ABB RobotStudio station: p2_celula_pick&place_R2022.rspag

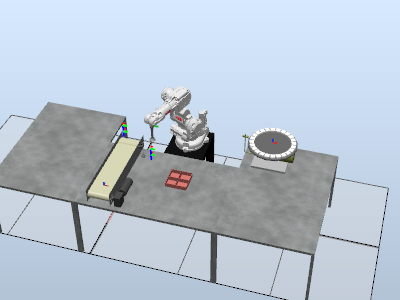
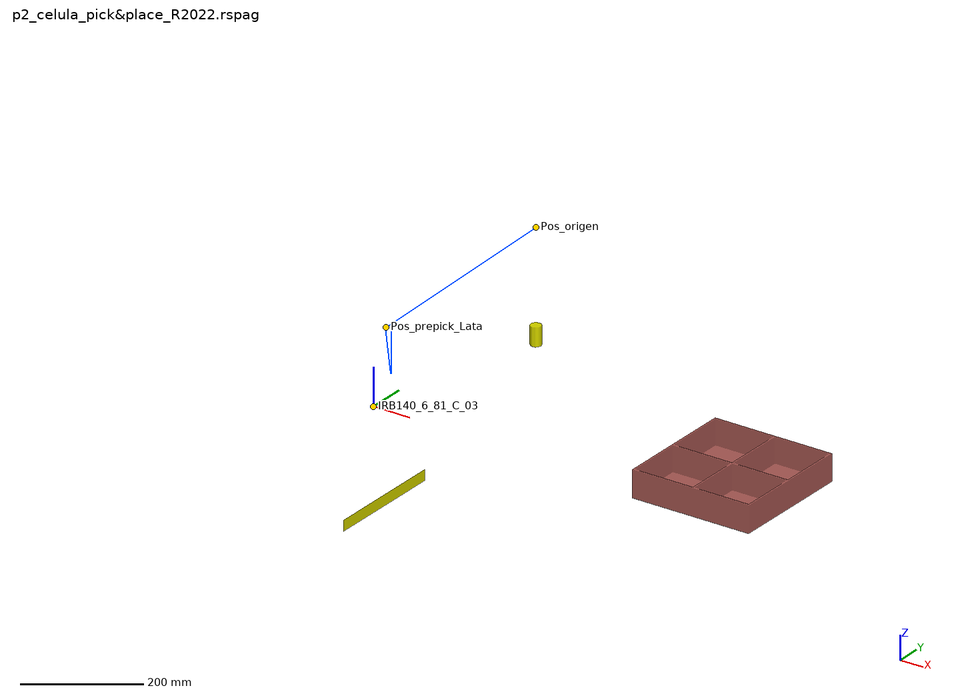
[picture v1: parts stored in the station drawn from their meshes, with robot base, taught points and paths (robot models come from the ABB library and are not in the file)]
--- station ---
Station p2_celula_cinta_mesagir_RS2019_2122_v2 (saved by RobotStudio 22.2.10013.1)
Controller Controlador1, task T_ROB1: task frame (RAPID world) sits at (-250, 750, 760) mm in the station
Controller Controlador1
  mechanical unit ROB_1: IRB140_6_81_C_03, 6 joints, base frame (0, 0, 0) mm
Layout (positions relative to the parent item):
  - Mesa de trabajo [part, from Project\Mesa de trabajo.rslib] at (1000, -110, 0) mm, rotated rx 0 ry 0 rz 90 deg
  - Soporte [part, from Project\SoporteDISA.rslib] at (-500, 970, 0) mm
  - Mesa giratoria [mechanism, from Project\CAD Mesa giratoria.rslib] at (-400, 1510, 760) mm; joint values [1.5268] (rad or m)
  - Mesa de trabajo_2 [part, from Project\Mesa de trabajo_2.rslib] at (1000, 2390, 0) mm, rotated rx 0 ry 0 rz 180 deg
  - cinta_transportadora [smart component, from Project\cinta_transportadoraDISA_RI_vf.rslib]
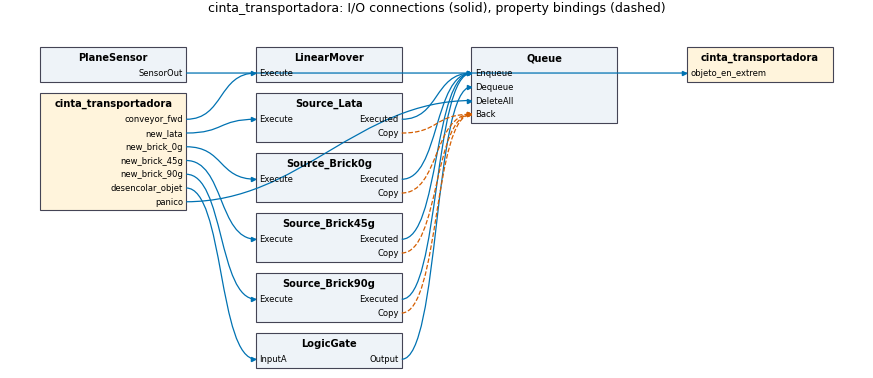
      connections:
        Source_Lata.Executed -> Queue.Enqueue
        PlaneSensor.SensorOut -> cinta_transportadora.objeto_en_extremo
        LogicGate.Output -> Queue.Dequeue
        cinta_transportadora.conveyor_fwd -> LinearMover.Execute
        cinta_transportadora.new_lata -> Source_Lata.Execute
        cinta_transportadora.new_brick_0g -> Source_Brick0g.Execute
        Source_Brick0g.Executed -> Queue.Enqueue
        cinta_transportadora.new_brick_45g -> Source_Brick45g.Execute
        Source_Brick45g.Executed -> Queue.Enqueue
        cinta_transportadora.new_brick_90g -> Source_Brick90g.Execute
        Source_Brick90g.Executed -> Queue.Enqueue
        cinta_transportadora.desencolar_objeto -> LogicGate.InputA
        cinta_transportadora.panico -> Queue.DeleteAll
        Source_Lata.Copy => Queue.Back
        Source_Brick0g.Copy => Queue.Back
        Source_Brick45g.Copy => Queue.Back
        Source_Brick90g.Copy => Queue.Back
    - Cinta transportadora [mechanism, from Project\CAD Cinta transportadora_2.rslib] at (940, 100, 865) mm, rotated rx 0 ry 0 rz 90 deg; joint values [0.66] (rad or m)
    - PlaneSensor [smart component, from Components\PlaneSensor.rslib]
        properties: Origin=[0.17366 0.29 0.93]; Axis1=[0 -0.23 0]; Axis2=[0 0 0.02]; SensedPart=(none)
      - _sensorPart_ [part], size 0 x 230 x 20 mm
    - Source_Lata [smart component, from Components\Source.rslib]
        properties: Source=lata_v3; Copy=(none); Parent=(none); Position=[0.9 0.175 0.9]; Orientation=[0 0 0]; Transient=false; PhysicsBehavior=0
    - Queue [smart component, from Components\Queue.rslib]
        properties: Back=(none); Front=(none); Queue={dff8c8d8-8fc0-4cec-b9db-be29e3a28473};{3f46c5cd-6d5b-48fe-86d8-48bb79a4d1fd};{fed15a07-9f68-4789-ad83-d232714e4fef};{72d5c8a9-7ca8-44e4-9c22-05c1b903e3c3};{2c04b273-edbc-4b62-af70-7d1944a2b1a7};{dd89b5b9-4857-4fa3-833c-eec227f403e2};{f4eddf35-6998-4428-b7c9-fa89e61066a5};{59d38785-21a3-4095-b70c-dd76d22c82fa};{f58c88b0-8b1a-4677-834d-2538b4835fbc};{bf0dbb8d-c78c-4188-b692-762c5a23a001};{d95e0b15-e936-410f-9e61-fe724db3c540};{2bd839ac-2019-415b-83b6-f6b4b81f6058};{944dfd5c-fb13-4575-94b9-afd36fb7f782};{83949a1e-8185-4c93-aa89-25b66602ceee};{4f3442c7-6ec6-4cb3-811a-33626f372c7a};{e17365bb-1bef-470b-b7e8-ca19aadd4809};{cf2dd58a-cd53-48dc-b704-49735820749d};{8950a759-9402-4139-8874-5414b657c79d};{ff666c08-3b55-4b31-af91-fb9ccf20597e};{00479655-b269-4748-adfd-ac0c9ff6814e};{97aee651-0048-42db-8271-c3c0405e84b6};{fb9d78cf-dec4-43c5-9643-90b43aa2c589};{1c737023-80b2-404b-b5f7-6a789b37bf94};{1ad73b80-f19d-4287-9cc4-3f5d513c44b3};{4a9cfcbd-6104-4fda-bb66-45b7a58cadba};{f5030ce7-8d9f-41fd-a0e0-943b87f40044};{6d643d8b-3f64-40eb-a316-e6579e800488};{a521ad28-28eb-4a02-9bff-ecd8140946c6};{54e7b961-4a7e-4eb9-9ad8-12fd860b0d09};{a76ff4cc-00e3-4c57-a249-5d676800b108};{a962051d-4321-485d-a7b6-d46c092dbce2};{12afaf56-49c6-4ccb-a620-f61642ea87b3};{899343f8-8cec-4edb-8463-23c64231605d};{4ef6d4c1-cd94-4d60-a742-53b60612dce5};{81835927-5480-4704-8e95-458aff66f5f4};{f557f8d3-d4c2-4ed9-81ee-a7371f7a9064};{a3283dab-8ae5-4a2f-a5f1-e3aa67324f00};{c73702e9-d765-4ca0-822f-348813278423};{414af213-d7ca-4e68-bc40-e9049d23ee9f};{a443fb2b-66d5-488a-b1cc-adbb6ebe2bc4};{96543467-7996-4e03-8609-ae8e4ea8f5a5};{8d69ce69-ef13-48be-9f25-6767b80184bb};{3789e405-e3ee-43e3-9d44-f2b54c75a36d};{dcf48f4d-3edb-45db-ad86-a5594296e2e2};{558120a7-5c88-4567-bb6c-c613c49afc30};{e83fdc9f-8db8-4194-8e9e-23232cbce353};{e901d7c8-de42-4474-a4d8-69454c384dc7};{2ec176ed-b9bc-4276-a128-5d5885d6c924};{8a74c292-b841-49af-a904-a0eec89b4ec6};{28ce9f31-519e-4f33-90fc-d50f408da8a6};{7a6d8f97-5379-4c1c-bdf6-f3c9a7aad7fa};{93e37ce4-f8bb-47c1-a0d2-06e10bf97d3f};{e8c5fbea-3965-4645-a5b7-c30112c44e96};{e7a5134e-a405-458e-8997-754f0378309b};{c78df5ee-6dfc-4a92-ba12-8dbc026209cf};{b1b4c00c-25a8-4bd7-80e1-6afde583105d};{dd0c4c06-6ce6-4be1-9c99-64db0c6bf6ff};{cefc24b7-ae8e-4a04-b8e7-f81f9433e3ae};{d6ce0fe5-35b2-42bb-b8d6-adbba0a8763d};{632131fa-8e51-4513-abd4-76a5ea6fcb33};{74bd1469-f266-4be2-92ac-ab91072705d8};{f6b76230-9575-465d-b1fa-b377b73fd13a};{9029fc77-8703-416f-ba68-5dca8c19555c};{b0ece3da-778c-4de5-ae49-5dd73d9e5191};{a4b8dd9f-1cea-46ee-b3db-e7479fcd6562};{ef382f55-caa7-4132-9e3f-cf775111e149};{7208aa9c-0a4c-4c08-824b-10d06152fb4f};{56b747bb-a3fb-4c38-b62b-aa802f47d477};{eb7448c0-cf7b-415d-9783-7e65fa723709};{f3dda0a0-cbf2-45ab-a7de-e8869eedcb74}; NumberOfObjects=0
    - LogicGate [smart component, from Components\LogicGate.rslib]
        properties: Operator=NOT; Delay=0
    - LinearMover [smart component, from Components\LinearMover.rslib]
        properties: Object=Queue; Direction=[1 0 0]; Speed=-0.1; Reference=Global; ReferenceObject=(none)
    - Source_Brick0g [smart component, from Components\Source.rslib]
        properties: Source=Brick0g; Copy=(none); Parent=(none); Position=[0.7 0.13 0.9]; Orientation=[0 0 0]; Transient=false; PhysicsBehavior=0
    - Source_Brick45g [smart component, from Components\Source.rslib]
        properties: Source=Brick0g; Copy=(none); Parent=(none); Position=[0.77 0.08 0.9]; Orientation=[0 0 0.785398163397448]; Transient=false; PhysicsBehavior=0
    - Source_Brick90g [smart component, from Components\Source.rslib]
        properties: Source=Brick0g; Copy=(none); Parent=(none); Position=[0.93 0.065 0.9]; Orientation=[0 0 1.5707963267949]; Transient=false; PhysicsBehavior=0
  - Pieza_11 [part], size 231 x 233 x 51.1 mm
  - Mesa de trabajo_3 [part, from Project\Mesa de trabajo_3.rslib] at (1000, -110, 0) mm, rotated rx 0 ry 0 rz 180 deg
  - ventosa_giu [smart component, from Project\ventosa_DISA_RI.rslib] at (245, 500, 1320) mm, rotated rx 180 ry 0 rz -180 deg
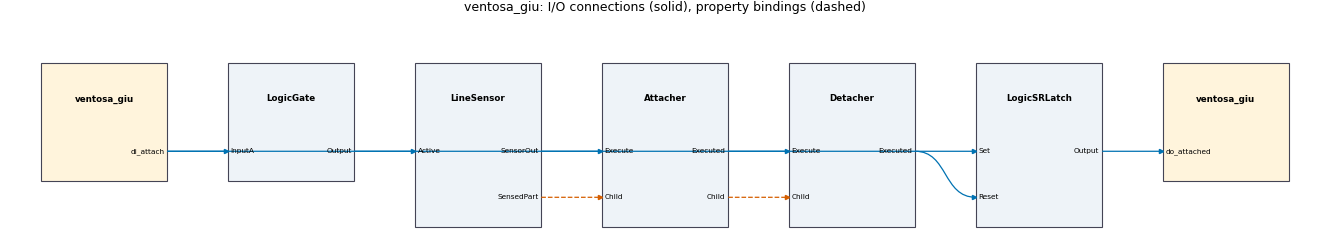
      connections:
        ventosa_giu.di_attach -> LogicGate.InputA
        LineSensor.SensorOut -> Attacher.Execute
        LogicGate.Output -> LineSensor.Active
        ventosa_giu.di_attach -> Detacher.Execute
        Attacher.Executed -> LogicSRLatch.Set
        Detacher.Executed -> LogicSRLatch.Reset
        LogicSRLatch.Output -> ventosa_giu.do_attached
        LineSensor.SensedPart => Attacher.Child
        Attacher.Child => Detacher.Child
    - ventosa_disa_giu [part, from Project\ventosa_DISA_RI.rslib]
    - LogicGate [smart component, from Components\LogicGate.rslib]
        properties: Operator=NOT; Delay=0
    - LineSensor [smart component, from Components\LineSensor.rslib]
        properties: Start=[0 0 0.175]; End=[0 0 0.21]; Radius=0.01; SensedPart=(none); SensedPoint=[0.337000091552734 0.776 0.848742248535156]
      - _sensorPart_ [part], size 20 x 20 x 35 mm
    - Attacher [smart component, from Components\Attacher.rslib]
        properties: Parent=ventosa_giu; Flange=0; Child=(none); Mount=false; Offset=[0 0 0]; Orientation=[0 0 0]
    - Detacher [smart component, from Components\Detacher.rslib]
        properties: Child=(none); KeepPosition=true
    - LogicSRLatch [smart component, from Components\LogicSRLatch.rslib]
  - IRB140_6_81_C_03 [mechanism, from Robots\IRB140_6_81_C_G_03.rslib] at (-250, 750, 760) mm; joint values [-0.4677, 0.3133, -0.1294, 0, 1.3869, -0.4677] (rad or m)
  - Brick0g [part], size 215 x 90 x 69 mm
  - lata_v3 [part], size 96.5 x 96.5 x 81.4 mm
Attachment: ventosa_giu is attached to IRB140_6_81_C_03 / Link6
EventTableEntry 9242: Group=, Trigger=Abrir 9243, Actions=[EventTableActionNothing 12035, EventTableActionDetach 12036, EventTableActionDetach 12037, EventTableActionDetach 12038, EventTableActionDetach 12039, EventTableActionDetach 12040, EventTableActionDetach 12041], Comment=, ActivationMode=2, Cyclic=true
EventTableTriggerIO 9243: IOValue=[1], IRC5Controller=? -1, Operator=0, SignalSource=? -1
EventTableEntry 9251: Group=, Trigger=Cerrar 9252, Actions=[EventTableActionDetach 12042, EventTableActionDetach 12043, EventTableActionDetach 12044, EventTableActionDetach 12045, EventTableActionDetach 12046, EventTableActionDetach 12047, EventTableActionNothing 12048], Comment=, ActivationMode=2, Cyclic=true
EventTableTriggerIO 9252: IOValue=[1], IRC5Controller=? -1, Operator=0, SignalSource=? -1
EventTableEntry 9264: Group=, Trigger=NOP 9265, Actions=[Abrir 9267], Comment=, ActivationMode=2, Cyclic=false
EventTableTriggerLogic 9265: Operand1=DoGARRAOPEN 9266, Operand2=? -1, Operator=4, Delay=1000
EventTableTriggerIO 9266: IOValue=[-1], IRC5Controller=? -1, Operator=0, SignalSource=? -1
EventTableActionIO 9267: IOValue=[-1], IRC5Controller=? -1, SignalTarget=? -1
EventTableEntry 9268: Group=, Trigger=NOT 9269, Actions=[Cerrar 9271], Comment=, ActivationMode=2, Cyclic=false
EventTableTriggerLogic 9269: layoutX=105, layoutY=91, Operand1=DoGARRAOPEN 9270, Operand2=? -1, Operator=2, Delay=1000
EventTableTriggerIO 9270: IOValue=[-1], IRC5Controller=? -1, Operator=0, SignalSource=? -1
EventTableActionIO 9271: IOValue=[-1], IRC5Controller=? -1, SignalTarget=? -1
EventTableEntry 9272: Group=, Trigger=DoGARRAOPEN 9273, Actions=[EventTableActionMechanicalPose 9274], Comment=, ActivationMode=2, Cyclic=false
EventTableTriggerIO 9273: IOValue=[1], IRC5Controller=? -1, Operator=0, SignalSource=? -1
EventTableActionMechanicalPose 9274: VirtualSignal=, Mechanism=? -1, ToPoseName=Abierta, VirtualSignalValue=[1]
EventTableEntry 9275: Group=, Trigger=DoGARRAOPEN 9276, Actions=[EventTableActionMechanicalPose 9277], Comment=, ActivationMode=2, Cyclic=false
EventTableTriggerIO 9276: IOValue=[0], IRC5Controller=? -1, Operator=0, SignalSource=? -1
EventTableActionMechanicalPose 9277: VirtualSignal=, Mechanism=? -1, ToPoseName=Cerrada, VirtualSignalValue=[1]
EventTableEntry 9288: Group=, Trigger=DO10_4 9289, Actions=[EventTableActionMechanicalPose 10691, EventTableActionMechanicalPose 10690, EventTableActionMechanicalPose 10689, EventTableActionMechanicalPose 11250, EventTableActionMechanicalPose 11251, EventTableActionMechanicalPose 11252], Comment=, ActivationMode=2, Cyclic=true
EventTableTriggerIO 9289: IOValue=[1], IRC5Controller=? -1, Operator=0, SignalSource=? -1
EventTableEntry 9711: Group=, Trigger=Abrir 9712, Actions=[EventTableActionNothing 12049, EventTableActionAttach 12050, EventTableActionAttach 12051, EventTableActionAttach 12052, EventTableActionNothing 12053, EventTableActionNothing 12054, EventTableActionNothing 12055], Comment=, ActivationMode=2, Cyclic=true
EventTableTriggerIO 9712: IOValue=[1], IRC5Controller=? -1, Operator=0, SignalSource=? -1
EventTableEntry 9938: Group=, Trigger=Cerrar 9939, Actions=[EventTableActionAttach 12056, EventTableActionAttach 12057, EventTableActionAttach 12058, EventTableActionAttach 12059, EventTableActionAttach 12060, EventTableActionAttach 12061, EventTableActionNothing 12062], Comment=, ActivationMode=2, Cyclic=true
EventTableTriggerIO 9939: IOValue=[1], IRC5Controller=? -1, Operator=0, SignalSource=? -1
EventTableActionMechanicalPose 10689: VirtualSignal=, Mechanism=Mesa giratoria 10339, ToPoseName=360º, VirtualSignalValue=[1]
EventTableActionMechanicalPose 10690: VirtualSignal=, Mechanism=Mesa giratoria 10339, ToPoseName=180º, VirtualSignalValue=[1]
EventTableActionMechanicalPose 10691: VirtualSignal=, Mechanism=Mesa giratoria 10339, ToPoseName=90º, VirtualSignalValue=[1]
EventTableEntry 11031: Group=, Trigger=DO10_5 11032, Actions=[EventTableActionAttach 11212, EventTableActionAttach 11213, EventTableActionAttach 11214], Comment=, ActivationMode=2, Cyclic=true
EventTableTriggerIO 11032: IOValue=[1], IRC5Controller=? -1, Operator=0, SignalSource=? -1
EventTableEntry 11051: Group=, Trigger=Abrir 11052, Actions=[EventTableActionNothing 12063, EventTableActionMechanicalPose 12064, EventTableActionMechanicalPose 12065, EventTableActionNothing 12066, EventTableActionNothing 12067, EventTableActionNothing 12068, EventTableActionNothing 12069], Comment=, ActivationMode=2, Cyclic=true
EventTableTriggerIO 11052: IOValue=[1], IRC5Controller=? -1, Operator=0, SignalSource=? -1
EventTableEntry 11203: Group=, Trigger=DO10_5 11204, Actions=[EventTableActionMechanicalPose 11205, EventTableActionMechanicalPose 11206, EventTableActionMechanicalPose 11207], Comment=, ActivationMode=2, Cyclic=true
EventTableTriggerIO 11204: IOValue=[1], IRC5Controller=? -1, Operator=0, SignalSource=? -1
EventTableActionMechanicalPose 11205: VirtualSignal=, Mechanism=Cinta transportadora 10989, ToPoseName=HomePosition, VirtualSignalValue=[1]
EventTableActionMechanicalPose 11206: VirtualSignal=, Mechanism=Cinta transportadora 10989, ToPoseName=HomePosition, VirtualSignalValue=[1]
EventTableActionMechanicalPose 11207: VirtualSignal=, Mechanism=Cinta transportadora 10989, ToPoseName=HomePosition, VirtualSignalValue=[1]
EventTableActionAttach 11212: AttachmentParent=Cinta transportadora 10989, AttachmentChild=? -1, MountObject=false, Offset=[X=1, Y=0, Z=0, W=0, X=0, Y=1, Z=0, W=0, X=0, Y=0, Z=1, W=0, X=0, Y=0, Z=0, W=1], FlangeIndext=0, FindNearest=false
EventTableActionAttach 11213: AttachmentParent=Cinta transportadora 10989, AttachmentChild=? -1, MountObject=false, Offset=[X=1, Y=0, Z=0, W=0, X=0, Y=1, Z=0, W=0, X=0, Y=0, Z=1, W=0, X=0, Y=0, Z=0, W=1], FlangeIndext=0, FindNearest=false
EventTableActionAttach 11214: AttachmentParent=Cinta transportadora 10989, AttachmentChild=? -1, MountObject=false, Offset=[X=1, Y=0, Z=0, W=0, X=0, Y=1, Z=0, W=0, X=0, Y=0, Z=1, W=0, X=0, Y=0, Z=0, W=1], FlangeIndext=0, FindNearest=false
EventTableActionMechanicalPose 11250: VirtualSignal=, Mechanism=Mesa giratoria 10339, ToPoseName=450, VirtualSignalValue=[1]
EventTableActionMechanicalPose 11251: VirtualSignal=, Mechanism=Mesa giratoria 10339, ToPoseName=540º, VirtualSignalValue=[1]
EventTableActionMechanicalPose 11252: VirtualSignal=, Mechanism=Mesa giratoria 10339, ToPoseName=SyncPosition, VirtualSignalValue=[1]
EventTableEntry 11270: Group=, Trigger=DO10_6 11271, Actions=[EventTableActionAttach 11272, EventTableActionAttach 11273, EventTableActionAttach 11274], Comment=, ActivationMode=2, Cyclic=true
EventTableTriggerIO 11271: IOValue=[1], IRC5Controller=? -1, Operator=0, SignalSource=? -1
EventTableActionAttach 11272: AttachmentParent=Cinta transportadora 10989, AttachmentChild=? -1, MountObject=false, Offset=[X=1, Y=0, Z=0, W=0, X=0, Y=1, Z=0, W=0, X=0, Y=0, Z=1, W=0, X=0, Y=0, Z=0, W=1], FlangeIndext=0, FindNearest=false
EventTableActionAttach 11273: AttachmentParent=Cinta transportadora 10989, AttachmentChild=? -1, MountObject=false, Offset=[X=1, Y=0, Z=0, W=0, X=0, Y=1, Z=0, W=0, X=0, Y=0, Z=1, W=0, X=0, Y=0, Z=0, W=1], FlangeIndext=0, FindNearest=false
EventTableActionAttach 11274: AttachmentParent=Cinta transportadora 10989, AttachmentChild=? -1, MountObject=false, Offset=[X=1, Y=0, Z=0, W=0, X=0, Y=1, Z=0, W=0, X=0, Y=0, Z=1, W=0, X=0, Y=0, Z=0, W=1], FlangeIndext=0, FindNearest=false
EventTableEntry 11487: Group=, Trigger=Cerrar 11488, Actions=[EventTableActionNothing 12070, EventTableActionNothing 12071, EventTableActionNothing 12072, EventTableActionNothing 12073, EventTableActionMechanicalPose 12074, EventTableActionMechanicalPose 12075, EventTableActionNothing 12076], Comment=, ActivationMode=2, Cyclic=true
EventTableTriggerIO 11488: IOValue=[1], IRC5Controller=? -1, Operator=0, SignalSource=? -1
EventTableEntry 11751: Group=, Trigger=Cerrar 11752, Actions=[EventTableActionNothing 12077, EventTableActionNothing 12078, EventTableActionNothing 12079, EventTableActionNothing 12080, EventTableActionDetach 12081, EventTableActionDetach 12082, EventTableActionDetach 12083], Comment=, ActivationMode=2, Cyclic=true
EventTableTriggerIO 11752: IOValue=[1], IRC5Controller=? -1, Operator=0, SignalSource=? -1
EventTableEntry 11847: Group=, Trigger=DO10_6 11848, Actions=[EventTableActionMechanicalPose 11849, EventTableActionMechanicalPose 11850, EventTableActionMechanicalPose 11851], Comment=, ActivationMode=2, Cyclic=true
EventTableTriggerIO 11848: IOValue=[1], IRC5Controller=? -1, Operator=0, SignalSource=? -1
EventTableActionMechanicalPose 11849: VirtualSignal=, Mechanism=Cinta transportadora 10989, ToPoseName=Final, VirtualSignalValue=[1]
EventTableActionMechanicalPose 11850: VirtualSignal=, Mechanism=Cinta transportadora 10989, ToPoseName=Final, VirtualSignalValue=[1]
EventTableActionMechanicalPose 11851: VirtualSignal=, Mechanism=Cinta transportadora 10989, ToPoseName=Final, VirtualSignalValue=[1]
EventTableActionNothing 12035: 
EventTableActionDetach 12036: AttachmentParent=? -1, AttachmentChild=? -1
EventTableActionDetach 12037: AttachmentParent=? -1, AttachmentChild=? -1
EventTableActionDetach 12038: AttachmentParent=? -1, AttachmentChild=? -1
EventTableActionDetach 12039: AttachmentParent=? -1, AttachmentChild=? -1
EventTableActionDetach 12040: AttachmentParent=? -1, AttachmentChild=? -1
EventTableActionDetach 12041: AttachmentParent=? -1, AttachmentChild=? -1
EventTableActionDetach 12042: AttachmentParent=Cinta transportadora 10989, AttachmentChild=? -1
EventTableActionDetach 12043: AttachmentParent=Cinta transportadora 10989, AttachmentChild=? -1
EventTableActionDetach 12044: AttachmentParent=Cinta transportadora 10989, AttachmentChild=? -1
EventTableActionDetach 12045: AttachmentParent=Mesa giratoria 10339, AttachmentChild=? -1
EventTableActionDetach 12046: AttachmentParent=Mesa giratoria 10339, AttachmentChild=? -1
EventTableActionDetach 12047: AttachmentParent=Mesa giratoria 10339, AttachmentChild=? -1
EventTableActionNothing 12048: 
EventTableActionNothing 12049: 
EventTableActionAttach 12050: AttachmentParent=Mesa giratoria 10339, AttachmentChild=? -1, MountObject=false, Offset=[X=1, Y=0, Z=0, W=0, X=0, Y=1, Z=0, W=0, X=0, Y=0, Z=1, W=0, X=0, Y=0, Z=0, W=1], FlangeIndext=0, FindNearest=false
EventTableActionAttach 12051: AttachmentParent=Mesa giratoria 10339, AttachmentChild=? -1, MountObject=false, Offset=[X=1, Y=0, Z=0, W=0, X=0, Y=1, Z=0, W=0, X=0, Y=0, Z=1, W=0, X=0, Y=0, Z=0, W=1], FlangeIndext=0, FindNearest=false
EventTableActionAttach 12052: AttachmentParent=Mesa giratoria 10339, AttachmentChild=? -1, MountObject=false, Offset=[X=1, Y=0, Z=0, W=0, X=0, Y=1, Z=0, W=0, X=0, Y=0, Z=1, W=0, X=0, Y=0, Z=0, W=1], FlangeIndext=0, FindNearest=false
EventTableActionNothing 12053: 
EventTableActionNothing 12054: 
EventTableActionNothing 12055: 
EventTableActionAttach 12056: AttachmentParent=? -1, AttachmentChild=? -1, MountObject=true, Offset=[X=1, Y=0, Z=0, W=0, X=0, Y=1, Z=0, W=0, X=0, Y=0, Z=1, W=0, X=0, Y=0, Z=0, W=1], FlangeIndext=0, FindNearest=false
EventTableActionAttach 12057: AttachmentParent=? -1, AttachmentChild=? -1, MountObject=true, Offset=[X=1, Y=0, Z=0, W=0, X=0, Y=1, Z=0, W=0, X=0, Y=0, Z=1, W=0, X=0, Y=0, Z=0, W=1], FlangeIndext=0, FindNearest=false
EventTableActionAttach 12058: AttachmentParent=? -1, AttachmentChild=? -1, MountObject=true, Offset=[X=1, Y=0, Z=0, W=0, X=0, Y=1, Z=0, W=0, X=0, Y=0, Z=1, W=0, X=0, Y=0, Z=0, W=1], FlangeIndext=0, FindNearest=false
EventTableActionAttach 12059: AttachmentParent=? -1, AttachmentChild=? -1, MountObject=true, Offset=[X=1, Y=0, Z=0, W=0, X=0, Y=1, Z=0, W=0, X=0, Y=0, Z=1, W=0, X=0, Y=0, Z=0, W=1], FlangeIndext=0, FindNearest=false
EventTableActionAttach 12060: AttachmentParent=? -1, AttachmentChild=? -1, MountObject=true, Offset=[X=1, Y=0, Z=0, W=0, X=0, Y=1, Z=0, W=0, X=0, Y=0, Z=1, W=0, X=0, Y=0, Z=0, W=1], FlangeIndext=0, FindNearest=false
EventTableActionAttach 12061: AttachmentParent=? -1, AttachmentChild=? -1, MountObject=true, Offset=[X=1, Y=0, Z=0, W=0, X=0, Y=1, Z=0, W=0, X=0, Y=0, Z=1, W=0, X=0, Y=0, Z=0, W=1], FlangeIndext=0, FindNearest=false
EventTableActionNothing 12062: 
EventTableActionNothing 12063: 
EventTableActionMechanicalPose 12064: VirtualSignal=, Mechanism=Cinta transportadora 10989, ToPoseName=Final_2, VirtualSignalValue=[1]
EventTableActionMechanicalPose 12065: VirtualSignal=, Mechanism=Cinta transportadora 10989, ToPoseName=Final_2, VirtualSignalValue=[1]
EventTableActionNothing 12066: 
EventTableActionNothing 12067: 
EventTableActionNothing 12068: 
EventTableActionNothing 12069: 
EventTableActionNothing 12070: 
EventTableActionNothing 12071: 
EventTableActionNothing 12072: 
EventTableActionNothing 12073: 
EventTableActionMechanicalPose 12074: VirtualSignal=, Mechanism=Cinta transportadora 10989, ToPoseName=Pose inicial_2, VirtualSignalValue=[1]
EventTableActionMechanicalPose 12075: VirtualSignal=, Mechanism=Cinta transportadora 10989, ToPoseName=Pose inicial_2, VirtualSignalValue=[1]
EventTableActionNothing 12076: 
EventTableActionNothing 12077: 
EventTableActionNothing 12078: 
EventTableActionNothing 12079: 
EventTableActionNothing 12080: 
EventTableActionDetach 12081: AttachmentParent=Cinta transportadora 10989, AttachmentChild=? -1
EventTableActionDetach 12082: AttachmentParent=Cinta transportadora 10989, AttachmentChild=? -1
EventTableActionDetach 12083: AttachmentParent=Cinta transportadora 10989, AttachmentChild=? -1
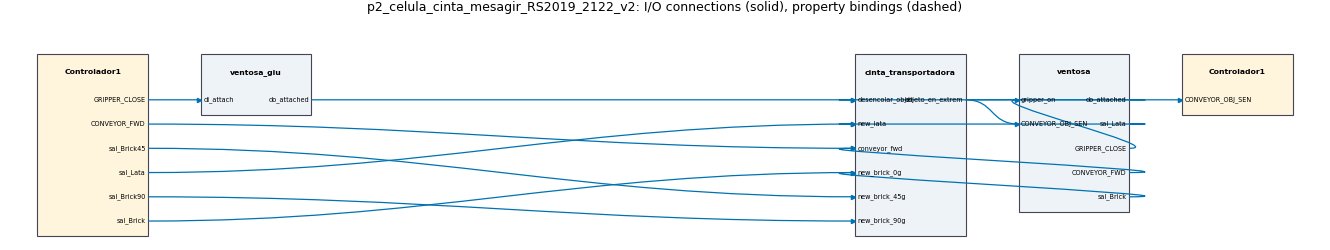
Station logic (signal -> signal, property => property):
  ventosa.do_attached -> cinta_transportadora.desencolar_objeto
  Controlador_P2_2021.sal_Lata -> cinta_transportadora.new_lata
  Controlador_P2_2021.GRIPPER_CLOSE -> ventosa.gripper_on
  cinta_transportadora.objeto_en_extremo -> Controlador_P2_2021.CONVEYOR_OBJ_SEN
  Controlador_P2_2021.CONVEYOR_FWD -> cinta_transportadora.conveyor_fwd
  Controlador_P2_2021.sal_Brick -> cinta_transportadora.new_brick_0g
  Controlador1.GRIPPER_CLOSE -> ventosa_giu.di_attach
  Controlador1.CONVEYOR_FWD -> cinta_transportadora.conveyor_fwd
  Controlador1.sal_Brick45 -> cinta_transportadora.new_brick_45g
  Controlador1.sal_Lata -> cinta_transportadora.new_lata
  Controlador1.sal_Brick90 -> cinta_transportadora.new_brick_90g
  Controlador1.sal_Brick -> cinta_transportadora.new_brick_0g
  cinta_transportadora.objeto_en_extremo -> Controlador1.CONVEYOR_OBJ_SEN
  ventosa_giu.do_attached -> cinta_transportadora.desencolar_objeto

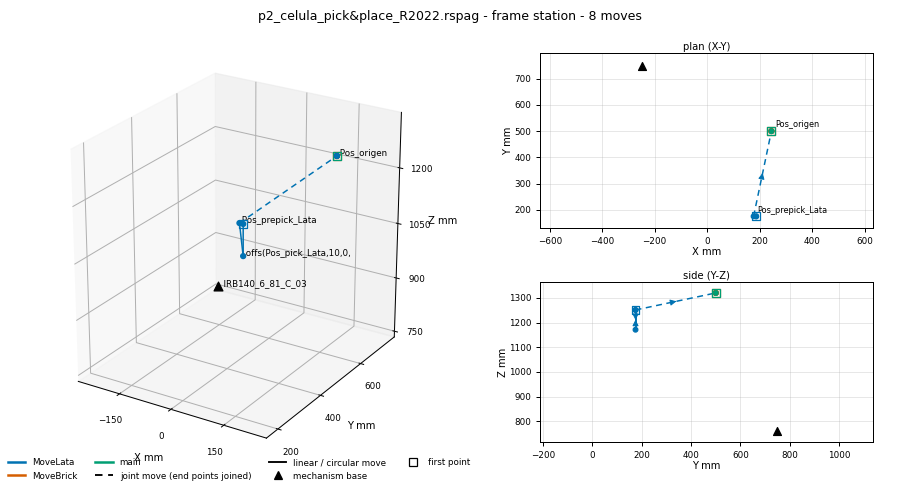
[picture p0: tool path of p2_celula_pick&place_R2022.rspag in frame station, 8 of 18 moves have a stored position in this frame; points joined in program order, loops and branches not executed]
--- Backups/Controlador1/RAPID/TASK1/PROGMOD/MainModule.mod ---
MODULE MainModule

    FUNC orient quatProd(orient o1, orient o2)


        RETURN [
            o1.q1 * o2.q1 - o1.q2 * o2.q2 - o1.q3 * o2.q3 - o1.q4 * o2.q4,
            o1.q1 * o2.q2 + o1.q2 * o2.q1 + o1.q3 * o2.q4 - o1.q4 * o2.q3,
            o1.q1 * o2.q3 + o1.q3 * o2.q1 + o1.q4 * o2.q2 - o1.q2 * o2.q4,
            o1.q1 * o2.q4 + o1.q4 * o2.q1 + o1.q2 * o2.q3 - o1.q3 * o2.q2];
    ENDFUNC


    PROC MoveLata(num latas,num layer)
        VAR robtarget preplace := Pos_preplace_lata;
        VAR robtarget place := Pos_place_lata;


        MoveL offs(Pos_prepick_Lata,10,0,0), v300, fine, tool0\WObj:=wobj0;
        MoveL offs(Pos_pick_Lata,10,0,0), v20, fine, tool0\WObj:=wobj0;
        Reset GRIPPER_CLOSE;
        MoveL Pos_prepick_Lata, v20, fine, tool0\WObj:=wobj0;
        MoveJ Pos_origen, v100, z100, tool0\WObj:=wobj0;


        preplace.trans.z := preplace.trans.z + 80*layer;
        place.trans.z := place.trans.z + 80*layer;

        TEST latas

        CASE 1:
            preplace.trans.x := preplace.trans.x + 115;
            place.trans.x := place.trans.x + 115;

        CASE 2:
            preplace.trans.x := preplace.trans.x + 115;
            place.trans.x := place.trans.x + 115;

            preplace.trans.y := preplace.trans.y + 115;
            place.trans.y := place.trans.y + 115;

        CASE 3:
             preplace.trans.y := preplace.trans.y + 115;
             place.trans.y := place.trans.y + 115;

        DEFAULT:
        ENDTEST

        MoveL preplace, v100, fine, tool0\WObj:=wobj0;
        MoveL place, v20, fine, tool0\WObj:=wobj0;

        Set GRIPPER_CLOSE;
        MoveL preplace, v20, fine, tool0\WObj:=wobj0;
        MoveL Pos_origen, v300, fine, tool0\WObj:=wobj0;

    ENDPROC



     PROC MoveBrick(num bricks, num angle)

        VAR robtarget prepick:=Pos_prepick_Brick;
        VAR robtarget pick:=Pos_pick_Brick;
        VAR robtarget preplace:=Pos_preplace_Brick;
        VAR robtarget place:=Pos_place_Brick;

        VAR orient oDef:=Pos_origen.rot;
        !VAR orient o45:=[0.92388,0,0,0.382];
        VAR orient on45:=[0.92388,0,0,-0.382];
        !VAR orient o90:=[0.7071,0,0,0.7071];
        VAR orient on90:=[0.7071,0,0,-0.7071];

        !o45:=quatProd(oDef,o45);
        on45:=quatProd(oDef,on45);
        !o90:=quatProd(oDef,o90);
        on90:=quatProd(oDef,on90);

        TEST angle
        CASE 45:
            prepick.rot:=on45;
            pick.rot:=on45;


            prepick.trans.x := prepick.trans.x + 15;
            pick.trans.x := pick.trans.x + 15;

            prepick.trans.y := prepick.trans.y - 20;
            pick.trans.y := pick.trans.y - 20;

        CASE 90:
            prepick.rot:=on90;
            pick.rot:=on90;

            prepick.trans.x := prepick.trans.x - 30;
            pick.trans.x := pick.trans.x - 30;

            prepick.trans.y := prepick.trans.y - 32;
            pick.trans.y := pick.trans.y - 32;

        DEFAULT:
            prepick.rot:=oDef;
            pick.rot:=oDef;
        ENDTEST

        MoveL prepick, v300, fine, tool0\WObj:=wobj0;
        MoveL pick, v20, fine, tool0\WObj:=wobj0;

        Reset GRIPPER_CLOSE;
        MoveL prepick, v20, fine, tool0\WObj:=wobj0;


        MoveJ Pos_origen, v100, z100, tool0\WObj:=wobj0;


        TEST bricks

        CASE 1:

            preplace.rot:=oDef;
            place.rot:=oDef;

            preplace.trans.y := preplace.trans.y + 105;
            place.trans.y := place.trans.y + 105;

        CASE 2:

            preplace.rot:=on90;
            place.rot:=on90;

            preplace.trans.z := preplace.trans.z + 60;
            place.trans.z := place.trans.z + 60;

            preplace.trans.x := preplace.trans.x + 21 - 180/2 + 90/2;
            place.trans.x := place.trans.x + 21 - 180/2 + 90/2;

            preplace.trans.y := preplace.trans.y + 90/2 + 15/2 - 21;
            place.trans.y := place.trans.y + 90/2 + 15/2 - 21;

        CASE 3:

            preplace.rot:=on90;
            place.rot:=on90;

            preplace.trans.z := preplace.trans.z + 60;
            place.trans.z := place.trans.z + 60;

            preplace.trans.x := preplace.trans.x + 21 - 180/2 + 90/2 + 15 + 90;
            place.trans.x := place.trans.x + 21 - 180/2 + 90/2 + 15 + 90;

            preplace.trans.y := preplace.trans.y + 90/2 + 15/2 - 21;
            place.trans.y := place.trans.y + 90/2 + 15/2 - 21;

        DEFAULT:
            preplace.rot:=oDef;
            place.rot:=oDef;
        ENDTEST


        MoveL preplace, v100, fine, tool0\WObj:=wobj0;
        MoveL place, v20, fine, tool0\WObj:=wobj0;
        Set GRIPPER_CLOSE;
        MoveL preplace, v20, fine, tool0\WObj:=wobj0;
        MoveL Pos_origen, v300, fine, tool0\WObj:=wobj0;
    ENDPROC





    PROC main()
        VAR num orientation := 0;
        VAR num bricks:=0;
        VAR num latas:=0;
        VAR num latas_layers:=0;

        BookErrNo NoSpaceError;


        set GRIPPER_CLOSE;
        MoveJ Pos_origen, v300, fine, tool0\WObj:=wobj0;

        Reset sal_Brick;
        Reset sal_Lata;


        WHILE TRUE DO
            Set CONVEYOR_FWD;


            IF sal_Brick = 1 THEN
                TPWrite "brick detected";
                IF bricks = 4 THEN
                    TPWrite "There is no space for bricks left!";
                    RAISE NoSpaceError;
                    RETURN;
                ENDIF

                orientation := 0;

                ReSet CONVEYOR_FWD;
                Set CONVEYOR_FWD;
                WaitDI CONVEYOR_OBJ_SEN, 1;
                Reset CONVEYOR_FWD;

                MoveBrick bricks, orientation;
                Reset sal_Brick;
                bricks := bricks+1;
            ENDIF

            IF sal_Brick45 = 1 THEN
                TPWrite "brick detected";
                IF bricks = 4 THEN
                    TPWrite "There is no space for bricks left!";
                    RAISE NoSpaceError;
                    RETURN;
                ENDIF

                orientation := 45;

                WaitDI CONVEYOR_OBJ_SEN, 1;
                Reset CONVEYOR_FWD;

                MoveBrick bricks, orientation;
                Reset sal_Brick45;
                bricks := bricks+1;
            ENDIF

            IF sal_Brick90 = 1 THEN
                TPWrite "brick detected";
                IF bricks = 4 THEN
                    TPWrite "There is no space for bricks left!";
                    RAISE NoSpaceError;
                    RETURN;
                ENDIF

                orientation :=90;

                WaitDI CONVEYOR_OBJ_SEN, 1;
                Reset CONVEYOR_FWD;

                MoveBrick bricks, orientation;
                Reset sal_Brick90;
                bricks := bricks+1;
            ENDIF

            IF sal_Lata = 1 THEN
                TPWrite "lata detected";
                IF latas_layers = 2 THEN
                    TPWrite "There is no space for latas left!";
                    RAISE NoSpaceError;
                    RETURN;
                ENDIF


                WaitDI CONVEYOR_OBJ_SEN, 1;
                Reset CONVEYOR_FWD;

                MoveLata latas,latas_layers;
                Reset sal_Lata;
                IF latas = 3 THEN
                    latas_layers := latas_layers+1;
                    latas:=0;
                ELSE
                    latas := latas+1;
                ENDIF
            ENDIF


            WaitTime 1;
        ENDWHILE
    ENDPROC


ENDMODULE

--- Backups/Controlador1/RAPID/TASK1/PROGMOD/Module1.mod ---
MODULE Module1
	CONST robtarget Pos_origen:=[[495,-250,560],[0,0,1,0],[-1,-1,-1,0],[9E+09,9E+09,9E+09,9E+09,9E+09,9E+09]];
	CONST robtarget Pos_prepick_Brick:=[[486,-578,484],[0,0,1,0],[-1,-1,-2,0],[9E+09,9E+09,9E+09,9E+09,9E+09,9E+09]];
	CONST robtarget Pos_pick_Brick:=[[486,-578,404],[0,0,1,0],[-1,-1,-2,0],[9E+09,9E+09,9E+09,9E+09,9E+09,9E+09]];
	CONST robtarget Pos_preplace_Brick:=[[610,-230,345],[0,0,1,0],[-1,-1,-1,0],[9E+09,9E+09,9E+09,9E+09,9E+09,9E+09]];
	CONST robtarget Pos_place_Brick:=[[610,-230,265.7],[0,0,1,0],[-1,-1,-1,0],[9E+09,9E+09,9E+09,9E+09,9E+09,9E+09]];
	CONST robtarget Pos_prepick_lata:=[[427,-575,491],[0,0,1,0],[-1,-1,-2,0],[9E+09,9E+09,9E+09,9E+09,9E+09,9E+09]];
	CONST robtarget Pos_pick_lata:=[[427,-575,411],[0,0,1,0],[-1,-1,-2,0],[9E+09,9E+09,9E+09,9E+09,9E+09,9E+09]];
	CONST robtarget Pos_preplace_lata:=[[587,26,360],[0,0,1,0],[0,-1,-1,0],[9E+09,9E+09,9E+09,9E+09,9E+09,9E+09]];
	CONST robtarget Pos_place_lata:=[[587,26,280],[0,0,1,0],[0,-1,-1,0],[9E+09,9E+09,9E+09,9E+09,9E+09,9E+09]];
    VAR errnum NoSpaceError:=-1;
ENDMODULE

--- Backups/Controlador1/SYSPAR/EIO.cfg ---
EIO:CFG_1.0:6:1::
#
EIO_CROSS:

      -Name "Lata" -Res "objeto_Lata" -Act1 "sal_Lata"

      -Name "Brick" -Res "objeto_Brick" -Act1 "sal_Brick"

      -Name "Brick45" -Res "objeto_Brick45" -Act1 "sal_Brick45"

      -Name "Brick90" -Res "objeto_Brick90" -Act1 "sal_Brick90"
#
EIO_SIGNAL:

      -Name "CONVEYOR_FWD" -SignalType "DO" -Access "All"

      -Name "CONVEYOR_BWD" -SignalType "DO" -Access "All"

      -Name "GRIPPER_CLOSE" -SignalType "DO" -Access "All"

      -Name "CONVEYOR_OBJ_SEN" -SignalType "DI" -Access "All"

      -Name "objeto_Lata" -SignalType "DI" -Access "All"

      -Name "objeto_Brick" -SignalType "DI" -Access "All"

      -Name "objeto_Brick45" -SignalType "DI" -Access "All"

      -Name "objeto_Brick90" -SignalType "DI" -Access "All"

      -Name "sal_Brick" -SignalType "DO" -Access "All"

      -Name "sal_Brick45" -SignalType "DO" -Access "All"

      -Name "sal_Brick90" -SignalType "DO" -Access "All"

      -Name "sal_Lata" -SignalType "DO" -Access "All"
